TYPE ST_StateMachine :
STRUCT
	uiInit 		: UINT;
	uiReady 	: UINT;
	uiBusy 		: UINT;
	uiWaiting 	: UINT;
	uiIdle 		: UINT;
	uiError 	: UINT;
END_STRUCT
END_TYPE

(* stored: Version 1.1.0.1, ProductVersion 3.1.4024.0
   DUT ST_StateMachine: Id {55662db1-7baf-4d79-8020-5daec45ea678} *)
